			IF CommandSTEP AND NOT CommandSTEPTRIG THEN
				TFCiclo_Deposito_Lastra_Depalettizzatore.Command_Step	:= TRUE;
				CommandSTEPTRIG := TRUE;
			ELSIF NOT CommandSTEP AND NOT CommandSTEPTRIG THEN
				TFCiclo_Deposito_Lastra_Depalettizzatore.Command_Step	:= FALSE;
				CommandSTEPTRIG := FALSE;
				CommandSTEP := FALSE;
			ELSIF  STEPCicloDONE THEN
				TFCiclo_Deposito_Lastra_Depalettizzatore.Command_Step	:= FALSE;
				CommandSTEP := FALSE;
				CommandSTEPTRIG := FALSE;
			END_IF
			
			TFCiclo_Deposito_Lastra_Depalettizzatore();
			STEPCicloDONE := TFCiclo_Deposito_Lastra_Depalettizzatore.STEPDone;
			
			IF Ciclo_Deposito_Lastra_Depal.Stato = TERMINATO THEN
				OUT.StartTilter := TRUE;
				ProductOnGripper := KNOPRODUCT;
				TFWorkFlowCase(ADR(WorkFlow[NumeroWF]),100,WorkflowCase_JMP);
			ELSIF (Ciclo_Deposito_Lastra_Depal.Stato = INTERROTTO AND (CmdExe.RapidStopRequest > 0 OR CmdExe.PhaseStopRequest > 0) AND Ciclo_Deposito_Lastra_Depal.Passo = 56 AND NOT OkDepositoDaLinea) THEN
				TFWorkFlowCase(ADR(WorkFlow[NumeroWF]),100,WorkflowCase_JMP);
			ELSIF Ciclo_Deposito_Lastra_Depal.Stato = INTERROTTO THEN	
				TFWorkFlowCase(ADR(WorkFlow[NumeroWF]),999,WorkflowCase_JMP);	
			END_IF

		(* Case 100 *)
		100:WorkFlow[NumeroWF].State := StateWF_END;
			WorkFlow[NumeroWF].Enable := FALSE;
			CommandSTEP := FALSE;
			CommandSTEPTRIG := FALSE;
			ResetComandoRibaltinoEseguito := FALSE;
			AssiInterpolati := FALSE;

		(* Case 999 *)
		(* WorkFlow ERROR *)
		StateWF_ERROR:
			TFWorkFlowError(ADR(WorkFlow[NumeroWF]),ADR(WorkFlowErrorLog[NumeroWF]));
			CmdExe.PhaseStopRequest := 1;
			CmdExe.RapidStopRequest := 1;
			WorkFlow[NumeroWF].Enable := FALSE;
			CommandSTEP := FALSE;
			CommandSTEPTRIG := FALSE;
			AssiInterpolati := FALSE;
		
		ELSE						
			TFWorkFlowError(ADR(WorkFlow[NumeroWF]),ADR(WorkFlowErrorLog[NumeroWF]));
			TFError(ErrNOCMDCASE,ErrNULL,ADR(CmdExe),ADR(State),ADR(Error),ADR(ErrorLog));	
	END_CASE;
END_IF
END_ACTION

END_FUNCTION_BLOCK

(* stored: Version 1.1.0.1, ProductVersion 3.1.4024.11
   POU TFMachinePalletizer_TF: Id {ce1a6238-33a3-4cee-9168-3b2637989b68}, SpecialFunc None
   Action WF02_CicloDiRiposo: Id {bc9c49a8-b0e9-4638-8487-3d24ed00159d}
   Action WF03_CicloPrelFalda: Id {b41d67c7-bad6-4721-b31b-51c2827b53fc}
   Action WF04_CicloDepFalda: Id {f3d3ade2-f8cf-4b84-b241-fc3f9de59c20}
   Action WF05_CicloPrelLastraDaPP: Id {b73d9e92-ce4d-433e-a661-c69732b17d5c}
   Action WF06_CicloDepLastraDaPP: Id {30fec531-b7d6-4a39-a8f9-a39de0bca3fc}
   Action WF07_CicloPrelLastraDaWA: Id {d2ec37b6-0813-4314-836a-5ea6dee9d3f6}
   Action WF08_CicloDepLastraSuPareggiatore: Id {8d83cd10-698b-49a1-bf08-1664c0ce72a5}
   Action WF09_CicloDepLastraDaWA: Id {f7133d13-13cc-4b52-87bb-c874bdd17301}
   Action WF10_CicloPelLastra_Depal: Id {9168d16d-10ac-4c5a-b75b-60b787d70133}
   Action WF11_CicloDepFalde_Depal: Id {489213be-aaf5-40a1-a2a2-bbb1da42fdbe}
   Action WF12_CicloDepLastra_Depal: Id {30866c03-294d-414c-b464-e0c9c9ac8599} *)
